(* CoDeSys 2.3 export: MARCHA_PARADA.EXP *)

(* POU Marcha_Parada, ST *)
PROGRAM Marcha_Parada
VAR_INPUT
	SFCReset:BOOL;
END_VAR
IEC_INITIAL_STEP Init:




END_STEP
(* @SFCMAXTIME := '' *)
(* @SFCMINTIME := '' *)
(* @SFCCOMMENT := '' *)
TRANSITION FROM Init TO Step2:= 
M


END_TRANSITION
IEC_STEP Step2:


Marcha(N);


END_STEP
(* @SFCMAXTIME := '' *)
(* @SFCMINTIME := '' *)
(* @SFCCOMMENT := '' *)
TRANSITION FROM Step2 TO Init:= 
Parada


END_TRANSITION
END_PROGRAM
